(* CoDeSys 2.3 export: RXQUEUE_10.EXP *)

(* Data type *)
TYPE RxQueue_10 :
STRUCT
	TxCounter      : UINT;
	RxCounter      : UINT;
	NoOfRxMessages : UINT;
	RxMessages     : ARRAY [0..9] OF ARRAY[0..13] OF BYTE;
END_STRUCT
END_TYPE
